{attribute 'qualified_only'}
{attribute 'strict'}
TYPE XY_Stage_State :
(
	off := 0,
	reset := 1,
	ready := 2,
	moving := 3,
	error := 9
);
END_TYPE

(* stored: Version 1.1.0.1, ProductVersion 3.1.4024.6
   DUT XY_Stage_State: Id {9036178f-97a3-4615-b4af-47bbe430ce8b} *)
